{attribute 'qualified_only'}
TYPE TrajectoryErrorCode :
(
	Undefined := 0,
  InvalidInput,
  SynchronizationFailed,
  CalculateStep1Failed
);
END_TYPE

(* stored: Version 1.1.0.1, ProductVersion 3.1.4024.9
   DUT TrajectoryErrorCode: Id {b6f9027e-b647-46b0-a8f4-fdacb3d850bf} *)
